// TIA Portal V17 export
// export: Created 2025-03-10T13:11:54.5717478Z, ExportSetting WithDefaults, DisplayName Totally Integrated Automation Portal, DisplayVersion V17 Update 8, DisplayName TIA Portal Openness, DisplayVersion V17 Update 8, DisplayName TIA Portal Version Control Interface, DisplayVersion V17, DisplayName SINAMICS Startdrive Advanced, DisplayVersion V17 SP2, DisplayName SINAMICS Startdrive G110M, G120, G120C, G120D, G120P, G115D, DisplayVersion V17 SP2, DisplayName SINAMICS Startdrive G130, G150, S120, S150, SINAMICS MV, S210, DisplayVersion V17 SP2, DisplayName STEP 7 Professional, DisplayVersion V17 Update 8, DisplayName SINUMERIK ONE STEP 7 Toolbox, DisplayVersion V17 Update 12, DisplayName SINUMERIK 840D sl STEP 7 Toolbox, DisplayVersion V17 Update 12, DisplayName STEP 7 Safety, DisplayVersion V17 Update 6, DisplayName WinCC Advanced, DisplayVersion V17 Update 8
TYPE "LBP_typeNC"
TITLE = NC interface / Interfaz CN / NC-Schnittstelle
// User data type for block LBP_NC [DB10] / Tipo de dato de usuario para bloque LBP_NC [DB10] / Anwender-Datentyp für Baustein LBP_NC [DB10]
// stored: IsFailsafeCompliant false
   STRUCT
      A_Disabl_Inp1 : Bool;   // Digitalen NCK-Eingang 1 deaktivieren / Disable digital NCK input 1 / Desactivar entrada digital NCK 1
      A_Disabl_Inp2 : Bool;   // Digitalen NCK-Eingang 2 deaktivieren / Disable digital NCK input 2 / Desactivar entrada digital NCK 2
      A_Disabl_Inp3 : Bool;   // Digitalen NCK-Eingang 3 deaktivieren / Disable digital NCK input 3 / Desactivar entrada digital NCK 3
      A_Disabl_Inp4 : Bool;   // Digitalen NCK-Eingang 4 deaktivieren / Disable digital NCK input 4 / Desactivar entrada digital NCK 4
      A_Disabl_Inp5 : Bool;   // Digitalen NCK-Eingang 5 deaktivieren / Disable digital NCK input 5 / Desactivar entrada digital NCK 5
      A_Disabl_Inp6 : Bool;   // Digitalen NCK-Eingang 6 deaktivieren / Disable digital NCK input 6 / Desactivar entrada digital NCK 6
      A_Disabl_Inp7 : Bool;   // Digitalen NCK-Eingang 7 deaktivieren / Disable digital NCK input 7 / Desactivar entrada digital NCK 7
      A_Disabl_Inp8 : Bool;   // Digitalen NCK-Eingang 8 deaktivieren / Disable digital NCK input 8 / Desactivar entrada digital NCK 8
      A_Set_Inp1 : Bool;   // Digitalen NCK-Eingang 1 setzen / Set digital NCK input 1 / Activar entrada digital NCK 1
      A_Set_Inp2 : Bool;   // Digitalen NCK-Eingang 2 setzen / Set digital NCK input 2 / Activar entrada digital NCK 2
      A_Set_Inp3 : Bool;   // Digitalen NCK-Eingang 3 setzen / Set digital NCK input 3 / Activar entrada digital NCK 3
      A_Set_Inp4 : Bool;   // Digitalen NCK-Eingang 4 setzen / Set digital NCK input 4 / Activar entrada digital NCK 4
      A_Set_Inp5 : Bool;   // Digitalen NCK-Eingang 5 setzen / Set digital NCK input 5 / Activar entrada digital NCK 5
      A_Set_Inp6 : Bool;   // Digitalen NCK-Eingang 6 setzen / Set digital NCK input 6 / Activar entrada digital NCK 6
      A_Set_Inp7 : Bool;   // Digitalen NCK-Eingang 7 setzen / Set digital NCK input 7 / Activar entrada digital NCK 7
      A_Set_Inp8 : Bool;   // Digitalen NCK-Eingang 8 setzen / Set digital NCK input 8 / Activar entrada digital NCK 8
      f0_f15 : Array[0..15] of Bool;   // Reserviert / Reserved / Reservado
      A_Disabl_Out1 : Bool;   // Digitalen NCK-Ausgang 1 deaktivieren / Disable digital NCK output 1 / Desactivar salida digital NCK 1
      A_Disabl_Out2 : Bool;   // Digitalen NCK-Ausgang 2 deaktivieren / Disable digital NCK output 2 / Desactivar salida digital NCK 2
      A_Disabl_Out3 : Bool;   // Digitalen NCK-Ausgang 3 deaktivieren / Disable digital NCK output 3 / Desactivar salida digital NCK 3
      A_Disabl_Out4 : Bool;   // Digitalen NCK-Ausgang 4 deaktivieren / Disable digital NCK output 4 / Desactivar salida digital NCK 4
      A_Disabl_Out5 : Bool;   // Digitalen NCK-Ausgang 5 deaktivieren / Disable digital NCK output 5 / Desactivar salida digital NCK 5
      A_Disabl_Out6 : Bool;   // Digitalen NCK-Ausgang 6 deaktivieren / Disable digital NCK output 6 / Desactivar salida digital NCK 6
      A_Disabl_Out7 : Bool;   // Digitalen NCK-Ausgang 7 deaktivieren / Disable digital NCK output 7 / Desactivar salida digital NCK 7
      A_Disabl_Out8 : Bool;   // Digitalen NCK-Ausgang 8 deaktivieren / Disable digital NCK output 8 / Desactivar salida digital NCK 8
      A_OvMask_Out1 : Bool;   // Maske von Digitalausgang 1 überschreiben / Overwrite mask of digital output 1 / Sobrescribir máscara de salida digital 1
      A_OvMask_Out2 : Bool;   // Maske von Digitalausgang 2 überschreiben / Overwrite mask of digital output 2 / Sobrescribir máscara de salida digital 2
      A_OvMask_Out3 : Bool;   // Maske von Digitalausgang 3 überschreiben / Overwrite mask of digital output 3 / Sobrescribir máscara de salida digital 3
      A_OvMask_Out4 : Bool;   // Maske von Digitalausgang 4 überschreiben / Overwrite mask of digital output 4 / Sobrescribir máscara de salida digital 4
      A_OvMask_Out5 : Bool;   // Maske von Digitalausgang 5 überschreiben / Overwrite mask of digital output 5 / Sobrescribir máscara de salida digital 5
      A_OvMask_Out6 : Bool;   // Maske von Digitalausgang 6 überschreiben / Overwrite mask of digital output 6 / Sobrescribir máscara de salida digital 6
      A_OvMask_Out7 : Bool;   // Maske von Digitalausgang 7 überschreiben / Overwrite mask of digital output 7 / Sobrescribir máscara de salida digital 7
      A_OvMask_Out8 : Bool;   // Maske von Digitalausgang 8 überschreiben / Overwrite mask of digital output 8 / Sobrescribir máscara de salida digital 8
      A_Set_Out1 : Bool;   // Digitalen NCK-Ausgang 1 setzen / Set digital NCK output 1 / Activar salida digital NCK 1
      A_Set_Out2 : Bool;   // Digitalen NCK-Ausgang 2 setzen / Set digital NCK output 2 / Activar salida digital NCK 2
      A_Set_Out3 : Bool;   // Digitalen NCK-Ausgang 3 setzen / Set digital NCK output 3 / Activar salida digital NCK 3
      A_Set_Out4 : Bool;   // Digitalen NCK-Ausgang 4 setzen / Set digital NCK output 4 / Activar salida digital NCK 4
      A_Set_Out5 : Bool;   // Digitalen NCK-Ausgang 5 setzen / Set digital NCK output 5 / Activar salida digital NCK 5
      A_Set_Out6 : Bool;   // Digitalen NCK-Ausgang 6 setzen / Set digital NCK output 6 / Activar salida digital NCK 6
      A_Set_Out7 : Bool;   // Digitalen NCK-Ausgang 7 setzen / Set digital NCK output 7 / Activar salida digital NCK 7
      A_Set_Out8 : Bool;   // Digitalen NCK-Ausgang 8 setzen / Set digital NCK output 8 / Activar salida digital NCK 8
      A_InMask_Out1 : Bool;   // Eingangsmaske von Digitalausgangt 1 / Input mask of digital output 1 / Máscara de entrada de la salida digital 1
      A_InMask_Out2 : Bool;   // Eingangsmaske von Digitalausgangt 2 / Input mask of digital output 2 / Máscara de entrada de la salida digital 2
      A_InMask_Out3 : Bool;   // Eingangsmaske von Digitalausgangt 3 / Input mask of digital output 3 / Máscara de entrada de la salida digital 3
      A_InMask_Out4 : Bool;   // Eingangsmaske von Digitalausgangt 4 / Input mask of digital output 4 / Máscara de entrada de la salida digital 4
      A_InMask_Out5 : Bool;   // Eingangsmaske von Digitalausgangt 5 / Input mask of digital output 5 / Máscara de entrada de la salida digital 5
      A_InMask_Out6 : Bool;   // Eingangsmaske von Digitalausgangt 6 / Input mask of digital output 6 / Máscara de entrada de la salida digital 6
      A_InMask_Out7 : Bool;   // Eingangsmaske von Digitalausgangt 7 / Input mask of digital output 7 / Máscara de entrada de la salida digital 7
      A_InMask_Out8 : Bool;   // Eingangsmaske von Digitalausgangt 8 / Input mask of digital output 8 / Máscara de entrada de la salida digital 8
      MCP1AxisTbl : Array[1..22] of Byte;   // Achsnummer Tabelle MCP1 / Axis number Table MCP1 / Número de eje tabla MCP1
      MCP1MaxAxis : Word;   // Max. Achsnr., muss kleiner sein als oder gleich LBP_ConfigData.MaxAxis / Max. of Axisno, must be smaller than or equal to LBP_ConfigData.MaxAxis / Máx. n.º de eje, debe ser menor o igual que LBP_ConfigData.MaxAxis
      MCP2AxisTbl : Array[1..22] of Byte;   // Achsnummer Tabelle MCP2 / Axis number Table MCP2 / Número de eje tabla MCP2
      MCP2MaxAxis : Word;   // Max. Achsnr., muss kleiner sein als oder gleich LBP_ConfigData.MaxAxis / Max. of Axisno, must be smaller than or equal to LBP_ConfigData.MaxAxis / Máx. n.º de eje, debe ser menor o igual que LBP_ConfigData.MaxAxis
      f56_0 : Bool;
      A_EMERGENCY : Bool;   // Not-Aus / Emergency stop / Parada de emergencia
      A_EMERGENCY_Ackn : Bool;   // Not-Aus quittieren / Acknowledge emergency stop / Confirmar parada de emergencia
      f56_3 : Bool;
      A_Keyswitch0 : Bool;   // Schlüsselschalter-Stellung 0 / Keyswitch position 0 / Posición 0 interruptor de llave
      A_Keyswitch1 : Bool;   // Schlüsselschalter-Stellung 1 / Keyswitch position 1 / Posición 1 interruptor de llave
      A_Keyswitch2 : Bool;   // Schlüsselschalter-Stellung 2 / Keyswitch position 2 / Posición 2 interruptor de llave
      A_Keyswitch3 : Bool;   // Schlüsselschalter-Stellung 3 / Keyswitch position 3 / Posición 3 interruptor de llave
      A_IncInModeGroup : Bool;   // NC-Eingänge in Betriebsartengruppenbereich aktiv / INC inputs in mode group range active / Entradas CN activas en rango de grupos de modos de operación
      f57_1 : Bool;
      f57_2 : Bool;
      A_PCshutdown : Bool;
      f57_4 : Bool;
      f57_5 : Bool;
      f57_6 : Bool;
      f57_7 : Bool;
      A_CA_DisableAutoMach : Bool;   // Kollisionsvermeidung deaktivieren: AUTO Maschine / Deactivate collision avoidance: AUTO Machine / Desactivar prevención de colisiones: máquina AUTO
      A_CA_DisableAutoTools : Bool;   // Kollisionsvermeidung deaktivieren: AUTO Werkzeuge / Deactivate collision avoidance: AUTO Tools / Desactivar prevención de colisiones: herramientas AUTO
      A_CA_DisableAutoWorkh : Bool;   // Kollisionsvermeidung deaktivieren: AUTO Werkstückhalter / Deactivate collision avoidance: AUTO Workholder / Desactivar prevención de colisiones: portapiezas AUTO
      A_CA_DisableAutoWorkp : Bool;   // Kollisionsvermeidung deaktivieren: AUTO Werkstücke / Deactivate collision avoidance: AUTO Workpieces / Desactivar prevención de colisiones: piezas AUTO
      A_CA_DisableJogMach : Bool;   // Kollisionsvermeidung deaktivieren: JOG Maschine / Deactivate collision avoidance: JOG Machine / Desactivar prevención de colisiones: máquina JOG
      A_CA_DisableJogTools : Bool;   // Kollisionsvermeidung deaktivieren: JOG Werkzeuge / Deactivate collision avoidance: JOG Tools / Desactivar prevención de colisiones: herramientas JOG
      A_CA_DisableJogWorkh : Bool;   // Kollisionsvermeidung deaktivieren: JOG Werkstückhalter / Deactivate collision avoidance: JOG Workholder / Desactivar prevención de colisiones: portapiezas JOG
      A_CA_DisableJogWorkp : Bool;   // Kollisionsvermeidung deaktivieren: JOG Werkstücke / Deactivate collision avoidance: JOG Workpieces / Desactivar prevención de colisiones: piezas JOG
      f59 : Byte;
      E_ActVal_In1 : Bool;   // Istwert von digitalem NCK-Onboard-Eingang 1 / Actual value of digital NCK onboard input 1 / Valor real de entrada digital integrada NCK 1
      E_ActVal_In2 : Bool;   // Istwert von digitalem NCK-Onboard-Eingang 2 / Actual value of digital NCK onboard input 2 / Valor real de entrada digital integrada NCK 2
      E_ActVal_In3 : Bool;   // Istwert von digitalem NCK-Onboard-Eingang 3 / Actual value of digital NCK onboard input 3 / Valor real de entrada digital integrada NCK 3
      E_ActVal_In4 : Bool;   // Istwert von digitalem NCK-Onboard-Eingang 4 / Actual value of digital NCK onboard input 4 / Valor real de entrada digital integrada NCK 4
      f60_4 : Bool;
      f60_5 : Bool;
      f60_6 : Bool;
      f60_7 : Bool;
      f61_f62 : Array[61..61] of Byte;
      E_Setpoint_Out1 : Bool;   // Sollwert von digitalem NCK-Ausgang 1 / Setpoint of digital NCK output 1 / Consigna de salida digital NCK 1
      E_Setpoint_Out2 : Bool;   // Sollwert von digitalem NCK-Ausgang 2 / Setpoint of digital NCK output 2 / Consigna de salida digital NCK 2
      E_Setpoint_Out3 : Bool;   // Sollwert von digitalem NCK-Ausgang 3 / Setpoint of digital NCK output 3 / Consigna de salida digital NCK 3
      E_Setpoint_Out4 : Bool;   // Sollwert von digitalem NCK-Ausgang 4 / Setpoint of digital NCK output 4 / Consigna de salida digital NCK 4
      E_Setpoint_Out5 : Bool;   // Sollwert von digitalem NCK-Ausgang 5 / Setpoint of digital NCK output 5 / Consigna de salida digital NCK 5
      E_Setpoint_Out6 : Bool;   // Sollwert von digitalem NCK-Ausgang 6 / Setpoint of digital NCK output 6 / Consigna de salida digital NCK 6
      E_Setpoint_Out7 : Bool;   // Sollwert von digitalem NCK-Ausgang 7 / Setpoint of digital NCK output 7 / Consigna de salida digital NCK 7
      E_Setpoint_Out8 : Bool;   // Sollwert von digitalem NCK-Ausgang 8 / Setpoint of digital NCK output 8 / Consigna de salida digital NCK 8
      f65_f67 : Array[65..66] of Byte;
      E_HW1_moved : Byte;   // Handrad 1 bewegt / Handwheel 1 moved / Volante 1 movido
      E_HW2_moved : Byte;   // Handrad 2 bewegt / Handwheel 2 moved / Volante 2 movido
      E_HW3_moved : Byte;   // Handrad 3 bewegt / Handwheel 3 moved / Volante 3 movido
      E_CounterInchMetr : Byte;   // Zähler ändern Zoll/metrische Einheiten / Change counter inch/metric system of units / Modificar contador pulgadas/unidades métricas
      E_MCP1AxisValid : Bool;   // Aus HT6 / From HT6 / Des HT6
      E_MCP1WCS : Bool;   // Aus HT6 / From HT6 / Des HT6
      f72_2 : Bool;
      f72_3 : Bool;
      f72_4 : Bool;
      f72_5 : Bool;
      f72_6 : Bool;
      E_MCP1AxKeyDisp : Bool;   // MCP1 Achstaste angezeigt / MCP1 Axis Key Displayed / Tecla de eje MCP1 mostrada
      E_MCP2AxisValid : Bool;   // Aus HT6 / From HT6 / Des HT6
      E_MCP2WCS : Bool;   // Aus HT6 / From HT6 / Des HT6
      f73_2 : Bool;
      f73_3 : Bool;
      f73_4 : Bool;
      f73_5 : Bool;
      f73_6 : Bool;
      E_MCP2AxKeyDisp : Bool;   // MCP2 Achstaste angezeigt / MCP2 Axis Key Displayed / Tecla de eje MCP2 mostrada
      MCP1AxisFromHMI : Array[1..6] of Byte;   // Achsnummer aus HT6 / Axis number from HT6 / Número de eje de HT6
      MCP2AxisFromHMI : Array[1..6] of Byte;   // Achsnummer aus HT6 / Axis number from HT6 / Número de eje de HT6
      res86 : Word;
      res88 : Byte;
      res89 : Byte;
      epsToPlc : Byte;
      epsFromPlc : Byte;
      MpiDpOk : Bool;   // Slaves am MPI/DP Ok / Slaves on MPI/DP Ok / Esclavos en MPI/DP OK
      DpOk : Bool;   // Slaves am DP OK / Slaves on DP Ok / Esclavos en DP OK
      PnOk : Bool;   // Slaves am PN Ok / Slaves on PN Ok / Esclavos en PN OK
      f92_3 : Bool;
      Disabl_AlarmMpiDp : Bool;   // Alarmmeldung "MPI/DP-Busfehler" deaktivieren(400551) / Disable alarm message "MPI/DP bus error" (400551) / Desactivar aviso de alarma "Error de bus MPI/DP" (400551)
      Disabl_AlarmDp : Bool;   // Alarmmeldung "DP-Busfehler" deaktivieren (400552) / Disable alarm message "DP bus error" (400552) / Desactivar aviso de alarma "Error de bus DP" (400552)
      Disabl_AlarmPn : Bool;   // Alarmmeldung "PN-Busfehler" deaktivieren(400553) / Disable alarm message "PN bus error" (400553) / Desactivar aviso de alarma "Error de bus PN" (400553)
      f92_7 : Bool;
      E_CA_DisableAutoMach : Bool;   // Kollisionsvermeidung deaktivieren: AUTO Maschine / Deactivate collision avoidance: AUTO Machine / Desactivar prevención de colisiones: máquina AUTO
      E_CA_DisableAutoTools : Bool;   // Kollisionsvermeidung deaktivieren: AUTO Werkzeuge / Deactivate collision avoidance: AUTO Tools / Desactivar prevención de colisiones: herramientas AUTO
      E_CA_DisableAutoWorkh : Bool;   // Kollisionsvermeidung deaktivieren: AUTO Werkstückhalter / Deactivate collision avoidance: AUTO Workholder / Desactivar prevención de colisiones: portapiezas AUTO
      E_CA_DisableAutoWorkp : Bool;   // Kollisionsvermeidung deaktivieren: AUTO Werkstücke / Deactivate collision avoidance: AUTO Workpieces / Desactivar prevención de colisiones: piezas AUTO
      E_CA_DisableJogMach : Bool;   // Kollisionsvermeidung deaktivieren: JOG Maschine / Deactivate collision avoidance: JOG Machine / Desactivar prevención de colisiones: máquina JOG
      E_CA_DisableJogTools : Bool;   // Kollisionsvermeidung deaktivieren: JOG Werkzeuge / Deactivate collision avoidance: JOG Tools / Desactivar prevención de colisiones: herramientas JOG
      E_CA_DisableJogWorkh : Bool;   // Kollisionsvermeidung deaktivieren: JOG Spannmittel / Disable collision avoidance: JOG Workholder / Deshabilitar prevención de colisiones: portapiezas JOG
      E_CA_DisableJogWorkp : Bool;   // Kollisionsvermeidung deaktivieren: JOG Werkstücke / Deactivate collision avoidance: JOG Workpieces / Desactivar prevención de colisiones: piezas JOG
      E_MCP1LostPackageWarn : Bool;   // Zeigt eine bevorstehende Trennung von MCP 1 an / Indicates an imminent disconnect of MCP 1 / Indica una desconexión inminente de MCP 1.
      E_MCP2LostPackageWarn : Bool;   // Zeigt eine bevorstehende Trennung von MCP 2 an / Indicates an imminent disconnect of MCP 2 / Indica una desconexión inminente de MCP 2.
      E_HTLostPackageWarn : Bool;   // Zeigt eine bevorstehende Trennung des Handheld Terminals an / Indicates an imminent disconnect of handheld terminal / Indica una desconexión inminente del terminal portátil.
      E_Op1KeyLostPackageWarn : Bool;   // Zeigt eine bevorstehende Trennung der direkten Tasten-Einheit 1 an / Indicates an imminent disconnect of direct key unit 1 / Indica una desconexión inminente de la unidad de teclas directas 1.
      E_Op2KeyLostPackageWarn : Bool;   // Zeigt eine bevorstehende Trennung der direkten Tasten-Einheit 2 an / Indicates an imminent disconnect of direct key unit 2 / Indica una desconexión inminente de la unidad de teclas directas 2.
      f94_5 : Bool;
      f94_6 : Bool;
      f94_7 : Bool;
      f95 : Byte;
      E_LanguageID : Byte;   // Sprachkennung am HMI / LanguageID on HMI / Identificador de idioma en HMI
      E_Chan_HW1_A : Bool;   // Kanalnummer für Handrad 1 A / Channel number for handwheel1 A / Número de canal para volante 1 A
      E_Chan_HW1_B : Bool;   // Kanalnummer für Handrad 1 B / Channel number for handwheel1 B / Número de canal para volante 1 B
      E_Chan_HW1_C : Bool;   // Kanalnummer für Handrad 1 C / Channel number for handwheel1 C / Número de canal para volante 1 C
      E_Chan_HW1_D : Bool;   // Kanalnummer für Handrad 1 D / Channel number for handwheel1 D / Número de canal para volante 1 D
      f97_4 : Bool;
      f97_5 : Bool;
      f97_6 : Bool;
      f97_7 : Bool;
      E_Chan_HW2_A : Bool;   // Kanalnummer für Handrad 2 A / Channel number for handwheel2 A / Número de canal para volante 2 A
      E_Chan_HW2_B : Bool;   // Kanalnummer für Handrad 2 B / Channel number for handwheel2 B / Número de canal para volante 2 B
      E_Chan_HW2_C : Bool;   // Kanalnummer für Handrad 2 C / Channel number for handwheel2 C / Número de canal para volante 2 C
      E_Chan_HW2_D : Bool;   // Kanalnummer für Handrad 2 D / Channel number for handwheel2 D / Número de canal para volante 2 D
      f98_4 : Bool;
      f98_5 : Bool;
      f98_6 : Bool;
      f98_7 : Bool;
      E_Chan_HW3_A : Bool;   // Kanalnummer für Handrad 3 A / Channel number for handwheel3 A / Número de canal para volante 3 A
      E_Chan_HW3_B : Bool;   // Kanalnummer für Handrad 3 B / Channel number for handwheel3 B / Número de canal para volante 3 B
      E_Chan_HW3_C : Bool;   // Kanalnummer für Handrad 3 C / Channel number for handwheel3 C / Número de canal para volante 3 C
      E_Chan_HW3_D : Bool;   // Kanalnummer für Handrad 3 D / Channel number for handwheel3 D / Número de canal para volante 3 D
      f99_4 : Bool;
      f99_5 : Bool;
      f99_6 : Bool;
      f99_7 : Bool;
      E_Ax_A_HW1 : Bool;   // Achsnummer für Handrad 1 A / Axis number for handwheel1 A / Número de eje para volante 1 A
      E_Ax_B_HW1 : Bool;   // Achsnummer für Handrad 1 B / Axis number for handwheel1 B / Número de eje para volante 1 B
      E_Ax_C_HW1 : Bool;   // Achsnummer für Handrad 1 C / Axis number for handwheel1 C / Número de eje para volante 1 C
      E_Ax_D_HW1 : Bool;   // Achsnummer für Handrad 1 D / Axis number for handwheel1 D / Número de eje para volante 1 D
      E_Ax_E_HW1 : Bool;   // Achsnummer für Handrad 1 E / Axis number for handwheel1 E / Número de eje para volante 1 E
      E_CHW_sel1 : Bool;   // Kontur-Handrad ausgewählt / Contour handwheel selected / Volante de contorno seleccionado
      E_HW_sel1 : Bool;   // Handrad ausgewählt / Handwheel selected / Volante seleccionado
      E_Mach_Ax1 : Bool;   // Maschinenachse / Machine axis / Eje de máquina
      E_Ax_A_HW2 : Bool;   // Achsnummer für Handrad 2 A / Axis number for handwheel2 A / Número de eje para volante 2 A
      E_Ax_B_HW2 : Bool;   // Achsnummer für Handrad 2 B / Axis number for handwheel2 B / Número de eje para volante 2 B
      E_Ax_C_HW2 : Bool;   // Achsnummer für Handrad 2 C / Axis number for handwheel2 C / Número de eje para volante 2 C
      E_Ax_D_HW2 : Bool;   // Achsnummer für Handrad 2 D / Axis number for handwheel2 D / Número de eje para volante 2 D
      E_Ax_E_HW2 : Bool;   // Achsnummer für Handrad 2 E / Axis number for handwheel2 E / Número de eje para volante 2 E
      E_CHW_sel2 : Bool;   // Kontur-Handrad ausgewählt / Contour handwheel selected / Volante de contorno seleccionado
      E_HW_sel2 : Bool;   // Handrad ausgewählt / Handwheel selected / Volante seleccionado
      E_Mach_Ax2 : Bool;   // Maschinenachse / Machine axis / Eje de máquina
      E_Ax_A_HW3 : Bool;   // Achsnummer für Handrad 3 A / Axis number for handwheel3 A / Número de eje para volante 3 A
      E_Ax_B_HW3 : Bool;   // Achsnummer für Handrad 3 B / Axis number for handwheel3 B / Número de eje para volante 3 B
      E_Ax_C_HW3 : Bool;   // Achsnummer für Handrad 3 C / Axis number for handwheel3 C / Número de eje para volante 3 C
      E_Ax_D_HW3 : Bool;   // Achsnummer für Handrad 3 D / Axis number for handwheel3 D / Número de eje para volante 3 D
      E_Ax_E_HW3 : Bool;   // Achsnummer für Handrad 3 E / Axis number for handwheel3 E / Número de eje para volante 3 E
      E_CHW_sel3 : Bool;   // Kontur-Handrad ausgewählt / Contour handwheel selected / Volante de contorno seleccionado
      E_HW_sel3 : Bool;   // Handrad ausgewählt / Handwheel selected / Volante seleccionado
      E_Mach_Ax3 : Bool;   // Maschinenachse / Machine axis / Eje de máquina
      E_RemDiag : Bool;   // Ferndiagnose / Remote Diagnostic / Diagnóstico remoto
      f103_1 : Bool;
      f103_2 : Bool;
      f103_3 : Bool;
      f103_4 : Bool;
      E_ATready : Bool;   // AT-Box bereit / AT box ready / Caja AT lista
      E_MMCTemp : Bool;   // HMI-Temperaturgrenze / HMI temperature limit / Límite de temperatura HMI
      E_MMCBatt : Bool;   // HMI 101/102 Batteriealarm / HMI 101/102 battery alarm / Alarma de batería HMI 101/102
      E_MCP1ready : Bool;   // MCP1 bereit / MCP1 ready / MCP1 listo
      E_MCP2ready : Bool;   // MCP2 bereit / MCP2 ready / MCP2 listo
      E_HTready : Bool;   // HT bereit / HT ready / HT listo
      E_Op1KeyReady : Bool;   // OP1 fertig / OP1 ready / OP1 listo
      E_Op2KeyReady : Bool;   // OP2 fertig / OP2 ready / OP2 listo
      f104_5 : Bool;
      E_FirstOB1 : Bool;   // Dieses Bit ist für den ersten OB1 Zyklus Ein / This bit is on for the first OB1 cycle / Este bit es para el primer ciclo OB1 Con
      E_NCKready : Bool;   // NCK CPU bereit / NCK CPU ready / NCK CPU lista
      E_CancelToolCmd : Bool;   // Abgebrochenen Werkzeugbefehl beenden / Terminate canceled tool command / Finalizar comando de herramienta cancelado
      f105_1 : Bool;
      f105_2 : Bool;
      f105_3 : Bool;
      f105_4 : Bool;
      f105_5 : Bool;
      f105_6 : Bool;
      f105_7 : Bool;
      E_CollCheckOff : Bool;   // Kollisionsprüfung Aus / Collisions check off / Comprobación de colisiones Des
      E_EMERGENCY : Bool;   // NOT-AUS aktiv / EMERGENCY STOP active / PARADA DE EMERGENCIA activa
      f106_2 : Bool;
      f106_3 : Bool;
      f106_4 : Bool;
      f106_5 : Bool;
      f106_6 : Bool;
      f106_7 : Bool;
      E_InspProbe1 : Bool;   // Messtaster 1 betätigt / Inspection probe 1 actuated / Palpador 1 accionado
      E_InspProbe2 : Bool;   // Messtaster 2 betätigt / Inspection probe 2 actuated / Palpador 2 accionado
      f107_2 : Bool;
      f107_3 : Bool;
      f107_4 : Bool;
      f107_5 : Bool;
      E_NCU_LinkActive : Bool;   // NCU-Verbindung aktiv / NCU link active / Conexión NCU activa
      E_SystemInchDim : Bool;   // System Zollmaße / System inch dimension / Sistema dimensiones en pulgadas
      f108_0 : Bool;
      E_MMC2Ready : Bool;   // MMC2-CPU bereit / MMC2-CPU ready / MMC2-CPU listo
      E_MMCMPIready : Bool;   // MMC1-CPU auf MPI bereit / MMC1-CPU on MPI ready / MMC1-CPU en MPI listo
      E_MMCBTSSready : Bool;   // MMC1-CPU auf BTSS bereit / MMC1-CPU on BTSS ready / MMC1-CPU en BTSS listo
      f108_4 : Bool;
      E_DrivesInCylOp : Bool;   // Antriebe im zyklischen Betrieb / Drives in cyclic operation / Accionamientos en funcionamiento cíclico
      E_611Dready : Bool;
      E_NCready : Bool;
      E_NCKalarm : Bool;   // NCK-Alarm steht an / NCK alarm present / Alarma NCK presente
      f109_1 : Bool;
      f109_2 : Bool;
      f109_3 : Bool;
      A_PC_OSfault : Bool;
      E_HTempAlarm : Bool;   // Kühlkörper-Temperaturalarm NCU 573 / Heat sink temperature alarm NCU 573 / Alarma temperatura disipador NCU 573
      E_ATempAlarm : Bool;   // Lufttemperatur-Alarm / Air temperature alarm / Alarma temperatura aire
      E_BattAlarm : Bool;   // NCK-Batteriealarm / NCK battery alarm / Alarma de batería NCK
      E_SWCamMinus : Array[0..31] of Bool;   // Software-Nocken minus [0..31] / Software cams minus [0..31] / Leva de software Menos [0..31]
      E_SWCamPlus : Array[0..31] of Bool;   // Software-Nocken plus [0..31] / Software cams plus [0..31] / Leva de software Más [0..31]
      f118_f121 : Array[0..3] of Byte;
      A_Disabl_Inp9 : Bool;   // Digitalen NCK-Eingang 9 deaktivieren / Disable digital NCK input 9 / Desactivar entrada digital NCK 9
      A_Disabl_Inp10 : Bool;   // Digitalen NCK-Eingang 10 deaktivieren / Disable digital NCK input 10 / Desactivar entrada digital NCK 10
      A_Disabl_Inp11 : Bool;   // Digitalen NCK-Eingang 11 deaktivieren / Disable digital NCK input 11 / Desactivar entrada digital NCK 11
      A_Disabl_Inp12 : Bool;   // Digitalen NCK-Eingang 12 deaktivieren / Disable digital NCK input 12 / Desactivar entrada digital NCK 12
      A_Disabl_Inp13 : Bool;   // Digitalen NCK-Eingang 13 deaktivieren / Disable digital NCK input 13 / Desactivar entrada digital NCK 13
      A_Disabl_Inp14 : Bool;   // Digitalen NCK-Eingang 14 deaktivieren / Disable digital NCK input 14 / Desactivar entrada digital NCK 14
      A_Disabl_Inp15 : Bool;   // Digitalen NCK-Eingang 15 deaktivieren / Disable digital NCK input 15 / Desactivar entrada digital NCK 15
      A_Disabl_Inp16 : Bool;   // Digitalen NCK-Eingang 16 deaktivieren / Disable digital NCK input 16 / Desactivar entrada digital NCK 16
      A_Set_Inp9 : Bool;   // Digitalen NCK-Eingang 9 setzen / Set digital NCK input 9 / Activar entrada digital NCK 9
      A_Set_Inp10 : Bool;   // Digitalen NCK-Eingang 10 setzen / Set digital NCK input 10 / Activar entrada digital NCK 10
      A_Set_Inp11 : Bool;   // Digitalen NCK-Eingang 11 setzen / Set digital NCK input 11 / Activar entrada digital NCK 11
      A_Set_Inp12 : Bool;   // Digitalen NCK-Eingang 12 setzen / Set digital NCK input 12 / Activar entrada digital NCK 12
      A_Set_Inp13 : Bool;   // Digitalen NCK-Eingang 13 setzen / Set digital NCK input 13 / Activar entrada digital NCK 13
      A_Set_Inp14 : Bool;   // Digitalen NCK-Eingang 14 setzen / Set digital NCK input 14 / Activar entrada digital NCK 14
      A_Set_Inp15 : Bool;   // Digitalen NCK-Eingang 15 setzen / Set digital NCK input 15 / Activar entrada digital NCK 15
      A_Set_Inp16 : Bool;   // Digitalen NCK-Eingang 16 setzen / Set digital NCK input 16 / Activar entrada digital NCK 16
      A_Disabl_Inp17 : Bool;   // Digitalen NCK-Eingang 17 deaktivieren / Disable digital NCK input 17 / Desactivar entrada digital NCK 17
      A_Disabl_Inp18 : Bool;   // Digitalen NCK-Eingang 18 deaktivieren / Disable digital NCK input 18 / Desactivar entrada digital NCK 18
      A_Disabl_Inp19 : Bool;   // Digitalen NCK-Eingang 19 deaktivieren / Disable digital NCK input 19 / Desactivar entrada digital NCK 19
      A_Disabl_Inp20 : Bool;   // Digitalen NCK-Eingang 20 deaktivieren / Disable digital NCK input 20 / Desactivar entrada digital NCK 20
      A_Disabl_Inp21 : Bool;   // Digitalen NCK-Eingang 21 deaktivieren / Disable digital NCK input 21 / Desactivar entrada digital NCK 21
      A_Disabl_Inp22 : Bool;   // Digitalen NCK-Eingang 22 deaktivieren / Disable digital NCK input 22 / Desactivar entrada digital NCK 22
      A_Disabl_Inp23 : Bool;   // Digitalen NCK-Eingang 23 deaktivieren / Disable digital NCK input 23 / Desactivar entrada digital NCK 23
      A_Disabl_Inp24 : Bool;   // Digitalen NCK-Eingang 24 deaktivieren / Disable digital NCK input 24 / Desactivar entrada digital NCK 24
      A_Set_Inp17 : Bool;   // Digitalen NCK-Eingang 17 setzen / Set digital NCK input 17 / Activar entrada digital NCK 17
      A_Set_Inp18 : Bool;   // Digitalen NCK-Eingang 18 setzen / Set digital NCK input 18 / Activar entrada digital NCK 18
      A_Set_Inp19 : Bool;   // Digitalen NCK-Eingang 19 setzen / Set digital NCK input 19 / Activar entrada digital NCK 19
      A_Set_Inp20 : Bool;   // Digitalen NCK-Eingang 20 setzen / Set digital NCK input 20 / Activar entrada digital NCK 20
      A_Set_Inp21 : Bool;   // Digitalen NCK-Eingang 21 setzen / Set digital NCK input 21 / Activar entrada digital NCK 21
      A_Set_Inp22 : Bool;   // Digitalen NCK-Eingang 22 setzen / Set digital NCK input 22 / Activar entrada digital NCK 22
      A_Set_Inp23 : Bool;   // Digitalen NCK-Eingang 23 setzen / Set digital NCK input 23 / Activar entrada digital NCK 23
      A_Set_Inp24 : Bool;   // Digitalen NCK-Eingang 24 setzen / Set digital NCK input 24 / Activar entrada digital NCK 24
      A_Disabl_Inp25 : Bool;   // Digitalen NCK-Eingang 25 deaktivieren / Disable digital NCK input 25 / Desactivar entrada digital NCK 25
      A_Disabl_Inp26 : Bool;   // Digitalen NCK-Eingang 26 deaktivieren / Disable digital NCK input 26 / Desactivar entrada digital NCK 26
      A_Disabl_Inp27 : Bool;   // Digitalen NCK-Eingang 27 deaktivieren / Disable digital NCK input 27 / Desactivar entrada digital NCK 27
      A_Disabl_Inp28 : Bool;   // Digitalen NCK-Eingang 28 deaktivieren / Disable digital NCK input 28 / Desactivar entrada digital NCK 28
      A_Disabl_Inp29 : Bool;   // Digitalen NCK-Eingang 29 deaktivieren / Disable digital NCK input 29 / Desactivar entrada digital NCK 29
      A_Disabl_Inp30 : Bool;   // Digitalen NCK-Eingang 30 deaktivieren / Disable digital NCK input 30 / Desactivar entrada digital NCK 30
      A_Disabl_Inp31 : Bool;   // Digitalen NCK-Eingang 31 deaktivieren / Disable digital NCK input 31 / Desactivar entrada digital NCK 31
      A_Disabl_Inp32 : Bool;   // Digitalen NCK-Eingang 32 deaktivieren / Disable digital NCK input 32 / Desactivar entrada digital NCK 32
      A_Set_Inp25 : Bool;   // Digitalen NCK-Eingang 25 setzen / Set digital NCK input 25 / Activar entrada digital NCK 25
      A_Set_Inp26 : Bool;   // Digitalen NCK-Eingang 26 setzen / Set digital NCK input 26 / Activar entrada digital NCK 26
      A_Set_Inp27 : Bool;   // Digitalen NCK-Eingang 27 setzen / Set digital NCK input 27 / Activar entrada digital NCK 27
      A_Set_Inp28 : Bool;   // Digitalen NCK-Eingang 28 setzen / Set digital NCK input 28 / Activar entrada digital NCK 28
      A_Set_Inp29 : Bool;   // Digitalen NCK-Eingang 29 setzen / Set digital NCK input 29 / Activar entrada digital NCK 29
      A_Set_Inp30 : Bool;   // Digitalen NCK-Eingang 30 setzen / Set digital NCK input 30 / Activar entrada digital NCK 30
      A_Set_Inp31 : Bool;   // Digitalen NCK-Eingang 31 setzen / Set digital NCK input 31 / Activar entrada digital NCK 31
      A_Set_Inp32 : Bool;   // Digitalen NCK-Eingang 32 setzen / Set digital NCK input 32 / Activar entrada digital NCK 32
      A_Disabl_Inp33 : Bool;   // Digitalen NCK-Eingang 33 deaktivieren / Disable digital NCK input 33 / Desactivar entrada digital NCK 33
      A_Disabl_Inp34 : Bool;   // Digitalen NCK-Eingang 34 deaktivieren / Disable digital NCK input 34 / Desactivar entrada digital NCK 34
      A_Disabl_Inp35 : Bool;   // Digitalen NCK-Eingang 35 deaktivieren / Disable digital NCK input 35 / Desactivar entrada digital NCK 35
      A_Disabl_Inp36 : Bool;   // Digitalen NCK-Eingang 36 deaktivieren / Disable digital NCK input 36 / Desactivar entrada digital NCK 36
      A_Disabl_Inp37 : Bool;   // Digitalen NCK-Eingang 37 deaktivieren / Disable digital NCK input 37 / Desactivar entrada digital NCK 37
      A_Disabl_Inp38 : Bool;   // Digitalen NCK-Eingang 38 deaktivieren / Disable digital NCK input 38 / Desactivar entrada digital NCK 38
      A_Disabl_Inp39 : Bool;   // Digitalen NCK-Eingang 39 deaktivieren / Disable digital NCK input 39 / Desactivar entrada digital NCK 39
      A_Disabl_Inp40 : Bool;   // Digitalen NCK-Eingang 40 deaktivieren / Disable digital NCK input 40 / Desactivar entrada digital NCK 40
      A_Set_Inp33 : Bool;   // Digitalen NCK-Eingang 33 setzen / Set digital NCK input 33 / Activar entrada digital NCK 33
      A_Set_Inp34 : Bool;   // Digitalen NCK-Eingang 34 setzen / Set digital NCK input 34 / Activar entrada digital NCK 34
      A_Set_Inp35 : Bool;   // Digitalen NCK-Eingang 35 setzen / Set digital NCK input 35 / Activar entrada digital NCK 35
      A_Set_Inp36 : Bool;   // Digitalen NCK-Eingang 36 setzen / Set digital NCK input 36 / Activar entrada digital NCK 36
      A_Set_Inp37 : Bool;   // Digitalen NCK-Eingang 37 setzen / Set digital NCK input 37 / Activar entrada digital NCK 37
      A_Set_Inp38 : Bool;   // Digitalen NCK-Eingang 38 setzen / Set digital NCK input 38 / Activar entrada digital NCK 38
      A_Set_Inp39 : Bool;   // Digitalen NCK-Eingang 39 setzen / Set digital NCK input 39 / Activar entrada digital NCK 39
      A_Set_Inp40 : Bool;   // Digitalen NCK-Eingang 40 setzen / Set digital NCK input 40 / Activar entrada digital NCK 40
      A_Disabl_Out9 : Bool;   // Digitalen NCK-Ausgang 9 deaktivieren / Disable digital NCK output 9 / Desactivar salida digital NCK 9
      A_Disabl_Out10 : Bool;   // Digitalen NCK-Ausgang 10 deaktivieren / Disable digital NCK output 10 / Desactivar salida digital NCK 10
      A_Disabl_Out11 : Bool;   // Digitalen NCK-Ausgang 11 deaktivieren / Disable digital NCK output 11 / Desactivar salida digital NCK 11
      A_Disabl_Out12 : Bool;   // Digitalen NCK-Ausgang 12 deaktivieren / Disable digital NCK output 12 / Desactivar salida digital NCK 12
      A_Disabl_Out13 : Bool;   // Digitalen NCK-Ausgang 13 deaktivieren / Disable digital NCK output 13 / Desactivar salida digital NCK 13
      A_Disabl_Out14 : Bool;   // Digitalen NCK-Ausgang 14 deaktivieren / Disable digital NCK output 14 / Desactivar salida digital NCK 14
      A_Disabl_Out15 : Bool;   // Digitalen NCK-Ausgang 15 deaktivieren / Disable digital NCK output 15 / Desactivar salida digital NCK 15
      A_Disabl_Out16 : Bool;   // Digitalen NCK-Ausgang 16 deaktivieren / Disable digital NCK output 16 / Desactivar salida digital NCK 16
      A_OvMask_Out9 : Bool;   // Maske von Digitalausgang 9 überschreiben / Overwrite mask of digital output 9 / Sobrescribir máscara de salida digital 9
      A_OvMask_Out10 : Bool;   // Maske von Digitalausgang 10 überschreiben / Overwrite mask of digital output 10 / Sobrescribir máscara de salida digital 10
      A_OvMask_Out11 : Bool;   // Maske von Digitalausgang 11 überschreiben / Overwrite mask of digital output 11 / Sobrescribir máscara de salida digital 11
      A_OvMask_Out12 : Bool;   // Maske von Digitalausgang 12 überschreiben / Overwrite mask of digital output 12 / Sobrescribir máscara de salida digital 12
      A_OvMask_Out13 : Bool;   // Maske von Digitalausgang 13 überschreiben / Overwrite mask of digital output 13 / Sobrescribir máscara de salida digital 13
      A_OvMask_Out14 : Bool;   // Maske von Digitalausgang 14 überschreiben / Overwrite mask of digital output 14 / Sobrescribir máscara de salida digital 14
      A_OvMask_Out15 : Bool;   // Maske von Digitalausgang 15 überschreiben / Overwrite mask of digital output 15 / Sobrescribir máscara de salida digital 15
      A_OvMask_Out16 : Bool;   // Maske von Digitalausgang 16 überschreiben / Overwrite mask of digital output 16 / Sobrescribir máscara de salida digital 16
      A_Set_Out9 : Bool;   // Digitalen NCK-Ausgang 9 setzen / Set digital NCK output 9 / Activar salida digital NCK 9
      A_Set_Out10 : Bool;   // Digitalen NCK-Ausgang 10 setzen / Set digital NCK output 10 / Activar salida digital NCK 10
      A_Set_Out11 : Bool;   // Digitalen NCK-Ausgang 11 setzen / Set digital NCK output 11 / Activar salida digital NCK 11
      A_Set_Out12 : Bool;   // Digitalen NCK-Ausgang 12 setzen / Set digital NCK output 12 / Activar salida digital NCK 12
      A_Set_Out13 : Bool;   // Digitalen NCK-Ausgang 13 setzen / Set digital NCK output 13 / Activar salida digital NCK 13
      A_Set_Out14 : Bool;   // Digitalen NCK-Ausgang 14 setzen / Set digital NCK output 14 / Activar salida digital NCK 14
      A_Set_Out15 : Bool;   // Digitalen NCK-Ausgang 15 setzen / Set digital NCK output 15 / Activar salida digital NCK 15
      A_Set_Out16 : Bool;   // Digitalen NCK-Ausgang 16 setzen / Set digital NCK output 16 / Activar salida digital NCK 16
      A_InMask_Out9 : Bool;   // Eingangsmaske von Digitalausgangt 9 / Input mask of digital output 9 / Máscara de entrada de la salida digital 9
      A_InMask_Out10 : Bool;   // Eingangsmaske von Digitalausgangt 10 / Input mask of digital output 10 / Máscara de entrada de la salida digital 10
      A_InMask_Out11 : Bool;   // Eingangsmaske von Digitalausgangt 11 / Input mask of digital output 11 / Máscara de entrada de la salida digital 11
      A_InMask_Out12 : Bool;   // Eingangsmaske von Digitalausgangt 12 / Input mask of digital output 12 / Máscara de entrada de la salida digital 12
      A_InMask_Out13 : Bool;   // Eingangsmaske von Digitalausgangt 13 / Input mask of digital output 13 / Máscara de entrada de la salida digital 13
      A_InMask_Out14 : Bool;   // Eingangsmaske von Digitalausgangt 14 / Input mask of digital output 14 / Máscara de entrada de la salida digital 14
      A_InMask_Out15 : Bool;   // Eingangsmaske von Digitalausgangt 15 / Input mask of digital output 15 / Máscara de entrada de la salida digital 15
      A_InMask_Out16 : Bool;   // Eingangsmaske von Digitalausgangt 16 / Input mask of digital output 16 / Máscara de entrada de la salida digital 16
      A_Disabl_Out17 : Bool;   // Digitalen NCK-Ausgang 17 deaktivieren / Disable digital NCK output 17 / Desactivar salida digital NCK 17
      A_Disabl_Out18 : Bool;   // Digitalen NCK-Ausgang 18 deaktivieren / Disable digital NCK output 18 / Desactivar salida digital NCK 18
      A_Disabl_Out19 : Bool;   // Digitalen NCK-Ausgang 19 deaktivieren / Disable digital NCK output 19 / Desactivar salida digital NCK 19
      A_Disabl_Out20 : Bool;   // Digitalen NCK-Ausgang 20 deaktivieren / Disable digital NCK output 20 / Desactivar salida digital NCK 20
      A_Disabl_Out21 : Bool;   // Digitalen NCK-Ausgang 21 deaktivieren / Disable digital NCK output 21 / Desactivar salida digital NCK 21
      A_Disabl_Out22 : Bool;   // Digitalen NCK-Ausgang 22 deaktivieren / Disable digital NCK output 22 / Desactivar salida digital NCK 22
      A_Disabl_Out23 : Bool;   // Digitalen NCK-Ausgang 23 deaktivieren / Disable digital NCK output 23 / Desactivar salida digital NCK 23
      A_Disabl_Out24 : Bool;   // Digitalen NCK-Ausgang 24 deaktivieren / Disable digital NCK output 24 / Desactivar salida digital NCK 24
      A_OvMask_Out17 : Bool;   // Maske von Digitalausgang 17 überschreiben / Overwrite mask of digital output 17 / Sobrescribir máscara de salida digital 17
      A_OvMask_Out18 : Bool;   // Maske von Digitalausgang 18 überschreiben / Overwrite mask of digital output 18 / Sobrescribir máscara de salida digital 18
      A_OvMask_Out19 : Bool;   // Maske von Digitalausgang 19 überschreiben / Overwrite mask of digital output 19 / Sobrescribir máscara de salida digital 19
      A_OvMask_Out20 : Bool;   // Maske von Digitalausgang 20 überschreiben / Overwrite mask of digital output 20 / Sobrescribir máscara de salida digital 20
      A_OvMask_Out21 : Bool;   // Maske von Digitalausgang 21 überschreiben / Overwrite mask of digital output 21 / Sobrescribir máscara de salida digital 21
      A_OvMask_Out22 : Bool;   // Maske von Digitalausgang 22 überschreiben / Overwrite mask of digital output 22 / Sobrescribir máscara de salida digital 22
      A_OvMask_Out23 : Bool;   // Maske von Digitalausgang 23 überschreiben / Overwrite mask of digital output 23 / Sobrescribir máscara de salida digital 23
      A_OvMask_Out24 : Bool;   // Maske von Digitalausgang 24 überschreiben / Overwrite mask of digital output 24 / Sobrescribir máscara de salida digital 24
      A_Set_Out17 : Bool;   // Digitalen NCK-Ausgang 17 setzen / Set digital NCK output 17 / Activar salida digital NCK 17
      A_Set_Out18 : Bool;   // Digitalen NCK-Ausgang 18 setzen / Set digital NCK output 18 / Activar salida digital NCK 18
      A_Set_Out19 : Bool;   // Digitalen NCK-Ausgang 19 setzen / Set digital NCK output 19 / Activar salida digital NCK 19
      A_Set_Out20 : Bool;   // Digitalen NCK-Ausgang 20 setzen / Set digital NCK output 20 / Activar salida digital NCK 20
      A_Set_Out21 : Bool;   // Digitalen NCK-Ausgang 21 setzen / Set digital NCK output 21 / Activar salida digital NCK 21
      A_Set_Out22 : Bool;   // Digitalen NCK-Ausgang 22 setzen / Set digital NCK output 22 / Activar salida digital NCK 22
      A_Set_Out23 : Bool;   // Digitalen NCK-Ausgang 23 setzen / Set digital NCK output 23 / Activar salida digital NCK 23
      A_Set_Out24 : Bool;   // Digitalen NCK-Ausgang 24 setzen / Set digital NCK output 24 / Activar salida digital NCK 24
      A_InMask_Out17 : Bool;   // Eingangsmaske von Digitalausgangt 17 / Input mask of digital output 17 / Máscara de entrada de la salida digital 17
      A_InMask_Out18 : Bool;   // Eingangsmaske von Digitalausgangt 18 / Input mask of digital output 18 / Máscara de entrada de la salida digital 18
      A_InMask_Out19 : Bool;   // Eingangsmaske von Digitalausgangt 19 / Input mask of digital output 19 / Máscara de entrada de la salida digital 19
      A_InMask_Out20 : Bool;   // Eingangsmaske von Digitalausgangt 20 / Input mask of digital output 20 / Máscara de entrada de la salida digital 20
      A_InMask_Out21 : Bool;   // Eingangsmaske von Digitalausgangt 21 / Input mask of digital output 21 / Máscara de entrada de la salida digital 21
      A_InMask_Out22 : Bool;   // Eingangsmaske von Digitalausgangt 22 / Input mask of digital output 22 / Máscara de entrada de la salida digital 22
      A_InMask_Out23 : Bool;   // Eingangsmaske von Digitalausgangt 23 / Input mask of digital output 23 / Máscara de entrada de la salida digital 23
      A_InMask_Out24 : Bool;   // Eingangsmaske von Digitalausgangt 24 / Input mask of digital output 24 / Máscara de entrada de la salida digital 24
      A_Disabl_Out25 : Bool;   // Digitalen NCK-Ausgang 25 deaktivieren / Disable digital NCK output 25 / Desactivar salida digital NCK 25
      A_Disabl_Out26 : Bool;   // Digitalen NCK-Ausgang 26 deaktivieren / Disable digital NCK output 26 / Desactivar salida digital NCK 26
      A_Disabl_Out27 : Bool;   // Digitalen NCK-Ausgang 27 deaktivieren / Disable digital NCK output 27 / Desactivar salida digital NCK 27
      A_Disabl_Out28 : Bool;   // Digitalen NCK-Ausgang 28 deaktivieren / Disable digital NCK output 28 / Desactivar salida digital NCK 28
      A_Disabl_Out29 : Bool;   // Digitalen NCK-Ausgang 29 deaktivieren / Disable digital NCK output 29 / Desactivar salida digital NCK 29
      A_Disabl_Out30 : Bool;   // Digitalen NCK-Ausgang 30 deaktivieren / Disable digital NCK output 30 / Desactivar salida digital NCK 30
      A_Disabl_Out31 : Bool;   // Digitalen NCK-Ausgang 31 deaktivieren / Disable digital NCK output 31 / Desactivar salida digital NCK 31
      A_Disabl_Out32 : Bool;   // Digitalen NCK-Ausgang 32 deaktivieren / Disable digital NCK output 32 / Desactivar salida digital NCK 32
      A_OvMask_Out25 : Bool;   // Maske von Digitalausgang 25 überschreiben / Overwrite mask of digital output 25 / Sobrescribir máscara de salida digital 25
      A_OvMask_Out26 : Bool;   // Maske von Digitalausgang 26 überschreiben / Overwrite mask of digital output 26 / Sobrescribir máscara de salida digital 26
      A_OvMask_Out27 : Bool;   // Maske von Digitalausgang 27 überschreiben / Overwrite mask of digital output 27 / Sobrescribir máscara de salida digital 27
      A_OvMask_Out28 : Bool;   // Maske von Digitalausgang 28 überschreiben / Overwrite mask of digital output 28 / Sobrescribir máscara de salida digital 28
      A_OvMask_Out29 : Bool;   // Maske von Digitalausgang 29 überschreiben / Overwrite mask of digital output 29 / Sobrescribir máscara de salida digital 29
      A_OvMask_Out30 : Bool;   // Maske von Digitalausgang 30 überschreiben / Overwrite mask of digital output 30 / Sobrescribir máscara de salida digital 30
      A_OvMask_Out31 : Bool;   // Maske von Digitalausgang 31 überschreiben / Overwrite mask of digital output 31 / Sobrescribir máscara de salida digital 31
      A_OvMask_Out32 : Bool;   // Maske von Digitalausgang 32 überschreiben / Overwrite mask of digital output 32 / Sobrescribir máscara de salida digital 32
      A_Set_Out25 : Bool;   // Digitalen NCK-Ausgang 25 setzen / Set digital NCK output 25 / Activar salida digital NCK 25
      A_Set_Out26 : Bool;   // Digitalen NCK-Ausgang 26 setzen / Set digital NCK output 26 / Activar salida digital NCK 26
      A_Set_Out27 : Bool;   // Digitalen NCK-Ausgang 27 setzen / Set digital NCK output 27 / Activar salida digital NCK 27
      A_Set_Out28 : Bool;   // Digitalen NCK-Ausgang 28 setzen / Set digital NCK output 28 / Activar salida digital NCK 28
      A_Set_Out29 : Bool;   // Digitalen NCK-Ausgang 29 setzen / Set digital NCK output 29 / Activar salida digital NCK 29
      A_Set_Out30 : Bool;   // Digitalen NCK-Ausgang 30 setzen / Set digital NCK output 30 / Activar salida digital NCK 30
      A_Set_Out31 : Bool;   // Digitalen NCK-Ausgang 31 setzen / Set digital NCK output 31 / Activar salida digital NCK 31
      A_Set_Out32 : Bool;   // Digitalen NCK-Ausgang 32 setzen / Set digital NCK output 32 / Activar salida digital NCK 32
      A_InMask_Out25 : Bool;   // Eingangsmaske von Digitalausgangt 25 / Input mask of digital output 25 / Máscara de entrada de la salida digital 25
      A_InMask_Out26 : Bool;   // Eingangsmaske von Digitalausgangt 26 / Input mask of digital output 26 / Máscara de entrada de la salida digital 26
      A_InMask_Out27 : Bool;   // Eingangsmaske von Digitalausgangt 27 / Input mask of digital output 27 / Máscara de entrada de la salida digital 27
      A_InMask_Out28 : Bool;   // Eingangsmaske von Digitalausgangt 28 / Input mask of digital output 28 / Máscara de entrada de la salida digital 28
      A_InMask_Out29 : Bool;   // Eingangsmaske von Digitalausgangt 29 / Input mask of digital output 29 / Máscara de entrada de la salida digital 29
      A_InMask_Out30 : Bool;   // Eingangsmaske von Digitalausgangt 30 / Input mask of digital output 30 / Máscara de entrada de la salida digital 30
      A_InMask_Out31 : Bool;   // Eingangsmaske von Digitalausgangt 31 / Input mask of digital output 31 / Máscara de entrada de la salida digital 31
      A_InMask_Out32 : Bool;   // Eingangsmaske von Digitalausgangt 32 / Input mask of digital output 32 / Máscara de entrada de la salida digital 32
      A_Disabl_Out33 : Bool;   // Digitalen NCK-Ausgang 33 deaktivieren / Disable digital NCK output 33 / Desactivar salida digital NCK 33
      A_Disabl_Out34 : Bool;   // Digitalen NCK-Ausgang 34 deaktivieren / Disable digital NCK output 34 / Desactivar salida digital NCK 34
      A_Disabl_Out35 : Bool;   // Digitalen NCK-Ausgang 35 deaktivieren / Disable digital NCK output 35 / Desactivar salida digital NCK 35
      A_Disabl_Out36 : Bool;   // Digitalen NCK-Ausgang 36 deaktivieren / Disable digital NCK output 36 / Desactivar salida digital NCK 36
      A_Disabl_Out37 : Bool;   // Digitalen NCK-Ausgang 37 deaktivieren / Disable digital NCK output 37 / Desactivar salida digital NCK 37
      A_Disabl_Out38 : Bool;   // Digitalen NCK-Ausgang 38 deaktivieren / Disable digital NCK output 38 / Desactivar salida digital NCK 38
      A_Disabl_Out39 : Bool;   // Digitalen NCK-Ausgang 39 deaktivieren / Disable digital NCK output 39 / Desactivar salida digital NCK 39
      A_Disabl_Out40 : Bool;   // Digitalen NCK-Ausgang 40 deaktivieren / Disable digital NCK output 40 / Desactivar salida digital NCK 40
      A_OvMask_Out33 : Bool;   // Maske von Digitalausgang 33 überschreiben / Overwrite mask of digital output 33 / Sobrescribir máscara de salida digital 33
      A_OvMask_Out34 : Bool;   // Maske von Digitalausgang 34 überschreiben / Overwrite mask of digital output 34 / Sobrescribir máscara de salida digital 34
      A_OvMask_Out35 : Bool;   // Maske von Digitalausgang 35 überschreiben / Overwrite mask of digital output 35 / Sobrescribir máscara de salida digital 35
      A_OvMask_Out36 : Bool;   // Maske von Digitalausgang 36 überschreiben / Overwrite mask of digital output 36 / Sobrescribir máscara de salida digital 36
      A_OvMask_Out37 : Bool;   // Maske von Digitalausgang 37 überschreiben / Overwrite mask of digital output 37 / Sobrescribir máscara de salida digital 37
      A_OvMask_Out38 : Bool;   // Maske von Digitalausgang 38 überschreiben / Overwrite mask of digital output 38 / Sobrescribir máscara de salida digital 38
      A_OvMask_Out39 : Bool;   // Maske von Digitalausgang 39 überschreiben / Overwrite mask of digital output 39 / Sobrescribir máscara de salida digital 39
      A_OvMask_Out40 : Bool;   // Maske von Digitalausgang 40 überschreiben / Overwrite mask of digital output 40 / Sobrescribir máscara de salida digital 40
      A_Set_Out33 : Bool;   // Digitalen NCK-Ausgang 33 setzen / Set digital NCK output 33 / Activar salida digital NCK 33
      A_Set_Out34 : Bool;   // Digitalen NCK-Ausgang 34 setzen / Set digital NCK output 34 / Activar salida digital NCK 34
      A_Set_Out35 : Bool;   // Digitalen NCK-Ausgang 35 setzen / Set digital NCK output 35 / Activar salida digital NCK 35
      A_Set_Out36 : Bool;   // Digitalen NCK-Ausgang 36 setzen / Set digital NCK output 36 / Activar salida digital NCK 36
      A_Set_Out37 : Bool;   // Digitalen NCK-Ausgang 37 setzen / Set digital NCK output 37 / Activar salida digital NCK 37
      A_Set_Out38 : Bool;   // Digitalen NCK-Ausgang 38 setzen / Set digital NCK output 38 / Activar salida digital NCK 38
      A_Set_Out39 : Bool;   // Digitalen NCK-Ausgang 39 setzen / Set digital NCK output 39 / Activar salida digital NCK 39
      A_Set_Out40 : Bool;   // Digitalen NCK-Ausgang 40 setzen / Set digital NCK output 40 / Activar salida digital NCK 40
      A_InMask_Out33 : Bool;   // Eingangsmaske von Digitalausgangt 33 / Input mask of digital output 33 / Máscara de entrada de la salida digital 33
      A_InMask_Out34 : Bool;   // Eingangsmaske von Digitalausgangt 34 / Input mask of digital output 34 / Máscara de entrada de la salida digital 34
      A_InMask_Out35 : Bool;   // Eingangsmaske von Digitalausgangt 35 / Input mask of digital output 35 / Máscara de entrada de la salida digital 35
      A_InMask_Out36 : Bool;   // Eingangsmaske von Digitalausgangt 36 / Input mask of digital output 36 / Máscara de entrada de la salida digital 36
      A_InMask_Out37 : Bool;   // Eingangsmaske von Digitalausgangt 37 / Input mask of digital output 37 / Máscara de entrada de la salida digital 37
      A_InMask_Out38 : Bool;   // Eingangsmaske von Digitalausgangt 38 / Input mask of digital output 38 / Máscara de entrada de la salida digital 38
      A_InMask_Out39 : Bool;   // Eingangsmaske von Digitalausgangt 39 / Input mask of digital output 39 / Máscara de entrada de la salida digital 39
      A_InMask_Out40 : Bool;   // Eingangsmaske von Digitalausgangt 40 / Input mask of digital output 40 / Máscara de entrada de la salida digital 40
      A_Disabl_anaIn1 : Bool;   // Analogen NCK-Eingang 1 deaktivieren / Disable analog NCK input 1 / Desactivar entrada analógica NCK 1
      A_Disabl_anaIn2 : Bool;   // Analogen NCK-Eingang 2 deaktivieren / Disable analog NCK input 2 / Desactivar entrada analógica NCK 2
      A_Disabl_anaIn3 : Bool;   // Analogen NCK-Eingang 3 deaktivieren / Disable analog NCK input 3 / Desactivar entrada analógica NCK 3
      A_Disabl_anaIn4 : Bool;   // Analogen NCK-Eingang 4 deaktivieren / Disable analog NCK input 4 / Desactivar entrada analógica NCK 4
      A_Disabl_anaIn5 : Bool;   // Analogen NCK-Eingang 5 deaktivieren / Disable analog NCK input 5 / Desactivar entrada analógica NCK 5
      A_Disabl_anaIn6 : Bool;   // Analogen NCK-Eingang 6 deaktivieren / Disable analog NCK input 6 / Desactivar entrada analógica NCK 6
      A_Disabl_anaIn7 : Bool;   // Analogen NCK-Eingang 7 deaktivieren / Disable analog NCK input 7 / Desactivar entrada analógica NCK 7
      A_Disabl_anaIn8 : Bool;   // Analogen NCK-Eingang 8 deaktivieren / Disable analog NCK input 8 / Desactivar entrada analógica NCK 8
      A_InMask_anaIn1 : Bool;   // Eingangsmaske des analogen NCK-Eingangs 1 / Input mask of analog NCK input 1 / Máscara de entrada de la entrada analógica del NCK 1
      A_InMask_anaIn2 : Bool;   // Eingangsmaske des analogen NCK-Eingangs 2 / Input mask of analog NCK input 2 / Máscara de entrada de la entrada analógica del NCK 2
      A_InMask_anaIn3 : Bool;   // Eingangsmaske des analogen NCK-Eingangs 3 / Input mask of analog NCK input 3 / Máscara de entrada de la entrada analógica del NCK 3
      A_InMask_anaIn4 : Bool;   // Eingangsmaske des analogen NCK-Eingangs 4 / Input mask of analog NCK input 4 / Máscara de entrada de la entrada analógica del NCK 4
      A_InMask_anaIn5 : Bool;   // Eingangsmaske des analogen NCK-Eingangs 5 / Input mask of analog NCK input 5 / Máscara de entrada de la entrada analógica del NCK 5
      A_InMask_anaIn6 : Bool;   // Eingangsmaske des analogen NCK-Eingangs 6 / Input mask of analog NCK input 6 / Máscara de entrada de la entrada analógica del NCK 6
      A_InMask_anaIn7 : Bool;   // Eingangsmaske des analogen NCK-Eingangs 7 / Input mask of analog NCK input 7 / Máscara de entrada de la entrada analógica del NCK 7
      A_InMask_anaIn8 : Bool;   // Eingangsmaske des analogen NCK-Eingangs 8 / Input mask of analog NCK input 8 / Máscara de entrada de la entrada analógica del NCK 8
      A_Setval_anaIn1 : Word;   // Wert von analogem NCK-Eingang 1 setzen / Set value of analog NCK input 1 / Activar valor de entrada analógica NCK 1
      A_Setval_anaIn2 : Word;   // Wert von analogem NCK-Eingang 2 setzen / Set value of analog NCK input 2 / Activar valor de entrada analógica NCK 2
      A_Setval_anaIn3 : Word;   // Wert von analogem NCK-Eingang 3 setzen / Set value of analog NCK input 3 / Activar valor de entrada analógica NCK 3
      A_Setval_anaIn4 : Word;   // Wert von analogem NCK-Eingang 4 setzen / Set value of analog NCK input 4 / Activar valor de entrada analógica NCK 4
      A_Setval_anaIn5 : Word;   // Wert von analogem NCK-Eingang 5 setzen / Set value of analog NCK input 5 / Activar valor de entrada analógica NCK 5
      A_Setval_anaIn6 : Word;   // Wert von analogem NCK-Eingang 6 setzen / Set value of analog NCK input 6 / Activar valor de entrada analógica NCK 6
      A_Setval_anaIn7 : Word;   // Wert von analogem NCK-Eingang 7 setzen / Set value of analog NCK input 7 / Activar valor de entrada analógica NCK 7
      A_Setval_anaIn8 : Word;   // Wert von analogem NCK-Eingang 8 setzen / Set value of analog NCK input 8 / Activar valor de entrada analógica NCK 8
      f164_f165 : Int;
      A_OvMask_anaOut1 : Bool;   // Maske von Analogausgang 1 überschreiben / Overwrite mask of analog output 1 / Sobrescribir máscara de salida analógica 1
      A_OvMask_anaOut2 : Bool;   // Maske von Analogausgang 2 überschreiben / Overwrite mask of analog output 2 / Sobrescribir máscara de salida analógica 2
      A_OvMask_anaOut3 : Bool;   // Maske von Analogausgang 3 überschreiben / Overwrite mask of analog output 3 / Sobrescribir máscara de salida analógica 3
      A_OvMask_anaOut4 : Bool;   // Maske von Analogausgang 4 überschreiben / Overwrite mask of analog output 4 / Sobrescribir máscara de salida analógica 4
      A_OvMask_anaOut5 : Bool;   // Maske von Analogausgang 5 überschreiben / Overwrite mask of analog output 5 / Sobrescribir máscara de salida analógica 5
      A_OvMask_anaOut6 : Bool;   // Maske von Analogausgang 6 überschreiben / Overwrite mask of analog output 6 / Sobrescribir máscara de salida analógica 6
      A_OvMask_anaOut7 : Bool;   // Maske von Analogausgang 7 überschreiben / Overwrite mask of analog output 7 / Sobrescribir máscara de salida analógica 7
      A_OvMask_anaOut8 : Bool;   // Maske von Analogausgang 8 überschreiben / Overwrite mask of analog output 8 / Sobrescribir máscara de salida analógica 8
      A_InMask_anaOut1 : Bool;   // Eingangsmaske des analogen NCK-Ausgangs 1 / Input mask of analog NCK output 1 / Máscara de entrada de la salida analógica del NCK 1
      A_InMask_anaOut2 : Bool;   // Eingangsmaske des analogen NCK-Ausgangs 2 / Input mask of analog NCK output 2 / Máscara de entrada de la salida analógica del NCK 2
      A_InMask_anaOut3 : Bool;   // Eingangsmaske des analogen NCK-Ausgangs 3 / Input mask of analog NCK output 3 / Máscara de entrada de la salida analógica del NCK 3
      A_InMask_anaOut4 : Bool;   // Eingangsmaske des analogen NCK-Ausgangs 4 / Input mask of analog NCK output 4 / Máscara de entrada de la salida analógica del NCK 4
      A_InMask_anaOut5 : Bool;   // Eingangsmaske des analogen NCK-Ausgangs 5 / Input mask of analog NCK output 5 / Máscara de entrada de la salida analógica del NCK 5
      A_InMask_anaOut6 : Bool;   // Eingangsmaske des analogen NCK-Ausgangs 6 / Input mask of analog NCK output 6 / Máscara de entrada de la salida analógica del NCK 6
      A_InMask_anaOut7 : Bool;   // Eingangsmaske des analogen NCK-Ausgangs 7 / Input mask of analog NCK output 7 / Máscara de entrada de la salida analógica del NCK 7
      A_InMask_anaOut8 : Bool;   // Eingangsmaske des analogen NCK-Ausgangs 8 / Input mask of analog NCK output 8 / Máscara de entrada de la salida analógica del NCK 8
      A_Disabl_anaOut1 : Bool;   // Analogen NCK-Ausgang 1 deaktivieren / Disable analog NCK output 1 / Desactivar salida analógica NCK 1
      A_Disabl_anaOut2 : Bool;   // Analogen NCK-Ausgang 2 deaktivieren / Disable analog NCK output 2 / Desactivar salida analógica NCK 2
      A_Disabl_anaOut3 : Bool;   // Analogen NCK-Ausgang 3 deaktivieren / Disable analog NCK output 3 / Desactivar salida analógica NCK 3
      A_Disabl_anaOut4 : Bool;   // Analogen NCK-Ausgang 4 deaktivieren / Disable analog NCK output 4 / Desactivar salida analógica NCK 4
      A_Disabl_anaOut5 : Bool;   // Analogen NCK-Ausgang 5 deaktivieren / Disable analog NCK output 5 / Desactivar salida analógica NCK 5
      A_Disabl_anaOut6 : Bool;   // Analogen NCK-Ausgang 6 deaktivieren / Disable analog NCK output 6 / Desactivar salida analógica NCK 6
      A_Disabl_anaOut7 : Bool;   // Analogen NCK-Ausgang 7 deaktivieren / Disable analog NCK output 7 / Desactivar salida analógica NCK 7
      A_Disabl_anaOut8 : Bool;   // Analogen NCK-Ausgang 8 deaktivieren / Disable analog NCK output 8 / Desactivar salida analógica NCK 8
      f169 : Byte;
      A_Setval_anaOut1 : Word;   // Wert von analogem NCK-Ausgang 1 setzen / Set value of analog NCK output 1 / Activar valor de salida analógica NCK 1
      A_Setval_anaOut2 : Word;   // Wert von analogem NCK-Ausgang 2 setzen / Set value of analog NCK output 2 / Activar valor de salida analógica NCK 2
      A_Setval_anaOut3 : Word;   // Wert von analogem NCK-Ausgang 3 setzen / Set value of analog NCK output 3 / Activar valor de salida analógica NCK 3
      A_Setval_anaOut4 : Word;   // Wert von analogem NCK-Ausgang 4 setzen / Set value of analog NCK output 4 / Activar valor de salida analógica NCK 4
      A_Setval_anaOut5 : Word;   // Wert von analogem NCK-Ausgang 5 setzen / Set value of analog NCK output 5 / Activar valor de salida analógica NCK 5
      A_Setval_anaOut6 : Word;   // Wert von analogem NCK-Ausgang 6 setzen / Set value of analog NCK output 6 / Activar valor de salida analógica NCK 6
      A_Setval_anaOut7 : Word;   // Wert von analogem NCK-Ausgang 7 setzen / Set value of analog NCK output 7 / Activar valor de salida analógica NCK 7
      A_Setval_anaOut8 : Word;   // Wert von analogem NCK-Ausgang 8 setzen / Set value of analog NCK output 8 / Activar valor de salida analógica NCK 8
      E_ActVal_In9 : Bool;   // Istwert von digitalem NCK-Eingang 9 / Actual value of digital NCK input 9 / Valor real de entrada digital NCK 9
      E_ActVal_In10 : Bool;   // Istwert von digitalem NCK-Eingang 10 / Actual value of digital NCK input 10 / Valor real de entrada digital NCK 10
      E_ActVal_In11 : Bool;   // Istwert von digitalem NCK-Eingang 11 / Actual value of digital NCK input 11 / Valor real de entrada digital NCK 11
      E_ActVal_In12 : Bool;   // Istwert von digitalem NCK-Eingang 12 / Actual value of digital NCK input 12 / Valor real de entrada digital NCK 12
      E_ActVal_In13 : Bool;   // Istwert von digitalem NCK-Eingang 13 / Actual value of digital NCK input 13 / Valor real de entrada digital NCK 13
      E_ActVal_In14 : Bool;   // Istwert von digitalem NCK-Eingang 14 / Actual value of digital NCK input 14 / Valor real de entrada digital NCK 14
      E_ActVal_In15 : Bool;   // Istwert von digitalem NCK-Eingang 15 / Actual value of digital NCK input 15 / Valor real de entrada digital NCK 15
      E_ActVal_In16 : Bool;   // Istwert von digitalem NCK-Eingang 16 / Actual value of digital NCK input 16 / Valor real de entrada digital NCK 16
      E_ActVal_In17 : Bool;   // Istwert von digitalem NCK-Eingang 17 / Actual value of digital NCK input 17 / Valor real de entrada digital NCK 17
      E_ActVal_In18 : Bool;   // Istwert von digitalem NCK-Eingang 18 / Actual value of digital NCK input 18 / Valor real de entrada digital NCK 18
      E_ActVal_In19 : Bool;   // Istwert von digitalem NCK-Eingang 19 / Actual value of digital NCK input 19 / Valor real de entrada digital NCK 19
      E_ActVal_In20 : Bool;   // Istwert von digitalem NCK-Eingang 20 / Actual value of digital NCK input 20 / Valor real de entrada digital NCK 20
      E_ActVal_In21 : Bool;   // Istwert von digitalem NCK-Eingang 21 / Actual value of digital NCK input 21 / Valor real de entrada digital NCK 21
      E_ActVal_In22 : Bool;   // Istwert von digitalem NCK-Eingang 22 / Actual value of digital NCK input 22 / Valor real de entrada digital NCK 22
      E_ActVal_In23 : Bool;   // Istwert von digitalem NCK-Eingang 23 / Actual value of digital NCK input 23 / Valor real de entrada digital NCK 23
      E_ActVal_In24 : Bool;   // Istwert von digitalem NCK-Eingang 24 / Actual value of digital NCK input 24 / Valor real de entrada digital NCK 24
      E_ActVal_In25 : Bool;   // Istwert von digitalem NCK-Eingang 25 / Actual value of digital NCK input 25 / Valor real de entrada digital NCK 25
      E_ActVal_In26 : Bool;   // Istwert von digitalem NCK-Eingang 26 / Actual value of digital NCK input 26 / Valor real de entrada digital NCK 26
      E_ActVal_In27 : Bool;   // Istwert von digitalem NCK-Eingang 27 / Actual value of digital NCK input 27 / Valor real de entrada digital NCK 27
      E_ActVal_In28 : Bool;   // Istwert von digitalem NCK-Eingang 28 / Actual value of digital NCK input 28 / Valor real de entrada digital NCK 28
      E_ActVal_In29 : Bool;   // Istwert von digitalem NCK-Eingang 29 / Actual value of digital NCK input 29 / Valor real de entrada digital NCK 29
      E_ActVal_In30 : Bool;   // Istwert von digitalem NCK-Eingang 30 / Actual value of digital NCK input 30 / Valor real de entrada digital NCK 30
      E_ActVal_In31 : Bool;   // Istwert von digitalem NCK-Eingang 31 / Actual value of digital NCK input 31 / Valor real de entrada digital NCK 31
      E_ActVal_In32 : Bool;   // Istwert von digitalem NCK-Eingang 32 / Actual value of digital NCK input 32 / Valor real de entrada digital NCK 32
      E_ActVal_In33 : Bool;   // Istwert von digitalem NCK-Eingang 33 / Actual value of digital NCK input 33 / Valor real de entrada digital NCK 33
      E_ActVal_In34 : Bool;   // Istwert von digitalem NCK-Eingang 34 / Actual value of digital NCK input 34 / Valor real de entrada digital NCK 34
      E_ActVal_In35 : Bool;   // Istwert von digitalem NCK-Eingang 35 / Actual value of digital NCK input 35 / Valor real de entrada digital NCK 35
      E_ActVal_In36 : Bool;   // Istwert von digitalem NCK-Eingang 36 / Actual value of digital NCK input 36 / Valor real de entrada digital NCK 36
      E_ActVal_In37 : Bool;   // Istwert von digitalem NCK-Eingang 37 / Actual value of digital NCK input 37 / Valor real de entrada digital NCK 37
      E_ActVal_In38 : Bool;   // Istwert von digitalem NCK-Eingang 38 / Actual value of digital NCK input 38 / Valor real de entrada digital NCK 38
      E_ActVal_In39 : Bool;   // Istwert von digitalem NCK-Eingang 39 / Actual value of digital NCK input 39 / Valor real de entrada digital NCK 39
      E_ActVal_In40 : Bool;   // Istwert von digitalem NCK-Eingang 40 / Actual value of digital NCK input 40 / Valor real de entrada digital NCK 40
      E_Setpoint_Out9 : Bool;   // Sollwert von digitalem NCK-Ausgang 9 / Setpoint of digital NCK output 9 / Consigna de salida digital NCK 9
      E_Setpoint_Out10 : Bool;   // Sollwert von digitalem NCK-Ausgang 10 / Setpoint of digital NCK output 10 / Consigna de salida digital NCK 10
      E_Setpoint_Out11 : Bool;   // Sollwert von digitalem NCK-Ausgang 11 / Setpoint of digital NCK output 11 / Consigna de salida digital NCK 11
      E_Setpoint_Out12 : Bool;   // Sollwert von digitalem NCK-Ausgang 12 / Setpoint of digital NCK output 12 / Consigna de salida digital NCK 12
      E_Setpoint_Out13 : Bool;   // Sollwert von digitalem NCK-Ausgang 13 / Setpoint of digital NCK output 13 / Consigna de salida digital NCK 13
      E_Setpoint_Out14 : Bool;   // Sollwert von digitalem NCK-Ausgang 14 / Setpoint of digital NCK output 14 / Consigna de salida digital NCK 14
      E_Setpoint_Out15 : Bool;   // Sollwert von digitalem NCK-Ausgang 15 / Setpoint of digital NCK output 15 / Consigna de salida digital NCK 15
      E_Setpoint_Out16 : Bool;   // Sollwert von digitalem NCK-Ausgang 16 / Setpoint of digital NCK output 16 / Consigna de salida digital NCK 16
      E_Setpoint_Out17 : Bool;   // Sollwert von digitalem NCK-Ausgang 17 / Setpoint of digital NCK output 17 / Consigna de salida digital NCK 17
      E_Setpoint_Out18 : Bool;   // Sollwert von digitalem NCK-Ausgang 18 / Setpoint of digital NCK output 18 / Consigna de salida digital NCK 18
      E_Setpoint_Out19 : Bool;   // Sollwert von digitalem NCK-Ausgang 19 / Setpoint of digital NCK output 19 / Consigna de salida digital NCK 19
      E_Setpoint_Out20 : Bool;   // Sollwert von digitalem NCK-Ausgang 20 / Setpoint of digital NCK output 20 / Consigna de salida digital NCK 20
      E_Setpoint_Out21 : Bool;   // Sollwert von digitalem NCK-Ausgang 21 / Setpoint of digital NCK output 21 / Consigna de salida digital NCK 21
      E_Setpoint_Out22 : Bool;   // Sollwert von digitalem NCK-Ausgang 22 / Setpoint of digital NCK output 22 / Consigna de salida digital NCK 22
      E_Setpoint_Out23 : Bool;   // Sollwert von digitalem NCK-Ausgang 23 / Setpoint of digital NCK output 23 / Consigna de salida digital NCK 23
      E_Setpoint_Out24 : Bool;   // Sollwert von digitalem NCK-Ausgang 24 / Setpoint of digital NCK output 24 / Consigna de salida digital NCK 24
      E_Setpoint_Out25 : Bool;   // Sollwert von digitalem NCK-Ausgang 25 / Setpoint of digital NCK output 25 / Consigna de salida digital NCK 25
      E_Setpoint_Out26 : Bool;   // Sollwert von digitalem NCK-Ausgang 26 / Setpoint of digital NCK output 26 / Consigna de salida digital NCK 26
      E_Setpoint_Out27 : Bool;   // Sollwert von digitalem NCK-Ausgang 27 / Setpoint of digital NCK output 27 / Consigna de salida digital NCK 27
      E_Setpoint_Out28 : Bool;   // Sollwert von digitalem NCK-Ausgang 28 / Setpoint of digital NCK output 28 / Consigna de salida digital NCK 28
      E_Setpoint_Out29 : Bool;   // Sollwert von digitalem NCK-Ausgang 29 / Setpoint of digital NCK output 29 / Consigna de salida digital NCK 29
      E_Setpoint_Out30 : Bool;   // Sollwert von digitalem NCK-Ausgang 30 / Setpoint of digital NCK output 30 / Consigna de salida digital NCK 30
      E_Setpoint_Out31 : Bool;   // Sollwert von digitalem NCK-Ausgang 31 / Setpoint of digital NCK output 31 / Consigna de salida digital NCK 31
      E_Setpoint_Out32 : Bool;   // Sollwert von digitalem NCK-Ausgang 32 / Setpoint of digital NCK output 32 / Consigna de salida digital NCK 32
      E_Setpoint_Out33 : Bool;   // Sollwert von digitalem NCK-Ausgang 33 / Setpoint of digital NCK output 33 / Consigna de salida digital NCK 33
      E_Setpoint_Out34 : Bool;   // Sollwert von digitalem NCK-Ausgang 34 / Setpoint of digital NCK output 34 / Consigna de salida digital NCK 34
      E_Setpoint_Out35 : Bool;   // Sollwert von digitalem NCK-Ausgang 35 / Setpoint of digital NCK output 35 / Consigna de salida digital NCK 35
      E_Setpoint_Out36 : Bool;   // Sollwert von digitalem NCK-Ausgang 36 / Setpoint of digital NCK output 36 / Consigna de salida digital NCK 36
      E_Setpoint_Out37 : Bool;   // Sollwert von digitalem NCK-Ausgang 37 / Setpoint of digital NCK output 37 / Consigna de salida digital NCK 37
      E_Setpoint_Out38 : Bool;   // Sollwert von digitalem NCK-Ausgang 38 / Setpoint of digital NCK output 38 / Consigna de salida digital NCK 38
      E_Setpoint_Out39 : Bool;   // Sollwert von digitalem NCK-Ausgang 39 / Setpoint of digital NCK output 39 / Consigna de salida digital NCK 39
      E_Setpoint_Out40 : Bool;   // Sollwert von digitalem NCK-Ausgang 40 / Setpoint of digital NCK output 40 / Consigna de salida digital NCK 40
      E_ActVal_anaIn1 : Word;   // Istwert von analogem NCK-Eingang 1 / Actual value of analog NCK input 1 / Valor real de entrada analógica NCK 1
      E_ActVal_anaIn2 : Word;   // Istwert von analogem NCK-Eingang 2 / Actual value of analog NCK input 2 / Valor real de entrada analógica NCK 2
      E_ActVal_anaIn3 : Word;   // Istwert von analogem NCK-Eingang 3 / Actual value of analog NCK input 3 / Valor real de entrada analógica NCK 3
      E_ActVal_anaIn4 : Word;   // Istwert von analogem NCK-Eingang 4 / Actual value of analog NCK input 4 / Valor real de entrada analógica NCK 4
      E_ActVal_anaIn5 : Word;   // Istwert von analogem NCK-Eingang 5 / Actual value of analog NCK input 5 / Valor real de entrada analógica NCK 5
      E_ActVal_anaIn6 : Word;   // Istwert von analogem NCK-Eingang 6 / Actual value of analog NCK input 6 / Valor real de entrada analógica NCK 6
      E_ActVal_anaIn7 : Word;   // Istwert von analogem NCK-Eingang 7 / Actual value of analog NCK input 7 / Valor real de entrada analógica NCK 7
      E_ActVal_anaIn8 : Word;   // Istwert von analogem NCK-Eingang 8 / Actual value of analog NCK input 8 / Valor real de entrada analógica NCK 8
      E_Setval_anaOut1 : Word;   // Wert von analogem NCK-Ausgang 1 setzen / Set value of analog NCK output 1 / Activar valor de salida analógica NCK 1
      E_Setval_anaOut2 : Word;   // Wert von analogem NCK-Ausgang 2 setzen / Set value of analog NCK output 2 / Activar valor de salida analógica NCK 2
      E_Setval_anaOut3 : Word;   // Wert von analogem NCK-Ausgang 3 setzen / Set value of analog NCK output 3 / Activar valor de salida analógica NCK 3
      E_Setval_anaOut4 : Word;   // Wert von analogem NCK-Ausgang 4 setzen / Set value of analog NCK output 4 / Activar valor de salida analógica NCK 4
      E_Setval_anaOut5 : Word;   // Wert von analogem NCK-Ausgang 5 setzen / Set value of analog NCK output 5 / Activar valor de salida analógica NCK 5
      E_Setval_anaOut6 : Word;   // Wert von analogem NCK-Ausgang 6 setzen / Set value of analog NCK output 6 / Activar valor de salida analógica NCK 6
      E_Setval_anaOut7 : Word;   // Wert von analogem NCK-Ausgang 7 setzen / Set value of analog NCK output 7 / Activar valor de salida analógica NCK 7
      E_Setval_anaOut8 : Word;   // Wert von analogem NCK-Ausgang 8 setzen / Set value of analog NCK output 8 / Activar valor de salida analógica NCK 8
      E_CollCheck : Array[0..7] of Byte;   // Kollisionsprüfung / Collisions check / Comprobación de colisiones
      A_CollCheck : Array[0..7] of Byte;   // Kollisionsprüfung / Collisions check / Comprobación de colisiones
      E_HW4_moved : Byte;   // Handrad 4 bewegt / Handwheel 4 moved / Volante 4 movido
      E_HW5_moved : Byte;   // Handrad 5 bewegt / Handwheel 5 moved / Volante 5 movido
      E_HW6_moved : Byte;   // Handrad 6 bewegt / Handwheel 6 moved / Volante 6 movido
      E_EHW1_stands : Bool;   // Ethernet-Handrad 1 in Ruhestellung / Ethernet handwheel 1 at rest / Volante Ethernet 1 en posición de reposo
      E_EHW2_stands : Bool;   // Ethernet-Handrad 2 in Ruhestellung / Ethernet handwheel 2 at rest / Volante Ethernet 2 en posición de reposo
      E_EHW3_stands : Bool;   // Ethernet-Handrad 3 in Ruhestellung / Ethernet handwheel 3 at rest / Volante Ethernet 3 en posición de reposo
      E_EHW4_stands : Bool;   // Ethernet-Handrad 4 in Ruhestellung / Ethernet handwheel 4 at rest / Volante Ethernet 4 en posición de reposo
      E_EHW5_stands : Bool;   // Ethernet-Handrad 5 in Ruhestellung / Ethernet handwheel 5 at rest / Volante Ethernet 5 en posición de reposo
      E_EHW6_stands : Bool;   // Ethernet-Handrad 6 in Ruhestellung / Ethernet handwheel 6 at rest / Volante Ethernet 6 en posición de reposo
      f245_6 : Bool;
      f245_7 : Bool;
      E_HMI_HW1Active : Bool;   // Handrad 1 aktiv / Handwheel 1 active / Volante 1 activo
      E_HMI_HW2Active : Bool;   // Handrad 2 aktiv / Handwheel 2 active / Volante 2 activo
      E_HMI_HW3Active : Bool;   // Handrad 3 aktiv / Handwheel 3 active / Volante 3 activo
      E_HMI_HW4Active : Bool;   // Handrad 4 aktiv / Handwheel 4 active / Volante 4 activo
      E_HMI_HW5Active : Bool;   // Handrad 5 aktiv / Handwheel 5 active / Volante 5 activo
      E_HMI_HW6Active : Bool;   // Handrad 6 aktiv / Handwheel 6 active / Volante 6 activo
      f246_6 : Bool;
      f246_7 : Bool;
      f247 : Byte;
      A_RobotStatus : Array[0..7] of Byte;   // Roboterstatus / Robot status / Estado de robot
      E_RobotControl : Array[0..7] of Byte;   // Robotersteuerung / Robot control / Control de robot
   END_STRUCT;
   // MCP1AxisTbl[1] := B#16#01;
   // MCP1AxisTbl[2] := B#16#02;
   // MCP1AxisTbl[3] := B#16#03;
   // MCP1AxisTbl[4] := B#16#04;
   // MCP1AxisTbl[5] := B#16#05;
   // MCP1AxisTbl[6] := B#16#06;
   // MCP1AxisTbl[7] := B#16#07;
   // MCP1AxisTbl[8] := B#16#08;
   // MCP1AxisTbl[9] := B#16#09;
   // MCP1AxisTbl[10] := B#16#0A;
   // MCP1AxisTbl[11] := B#16#0B;
   // MCP1AxisTbl[12] := B#16#0C;
   // MCP2AxisTbl[1] := B#16#01;
   // MCP2AxisTbl[2] := B#16#02;
   // MCP2AxisTbl[3] := B#16#03;
   // MCP2AxisTbl[4] := B#16#04;
   // MCP2AxisTbl[5] := B#16#05;
   // MCP2AxisTbl[6] := B#16#06;
   // MCP2AxisTbl[7] := B#16#07;
   // MCP2AxisTbl[8] := B#16#08;
   // MCP2AxisTbl[9] := B#16#09;
   // MCP2AxisTbl[10] := B#16#0A;
   // MCP2AxisTbl[11] := B#16#0B;
   // MCP2AxisTbl[12] := B#16#0C;
END_TYPE
